FUNCTION_BLOCK HVAC_B28_Main_Seq
VAR_INPUT
END_VAR
VAR_OUTPUT
END_VAR
VAR
END_VAR

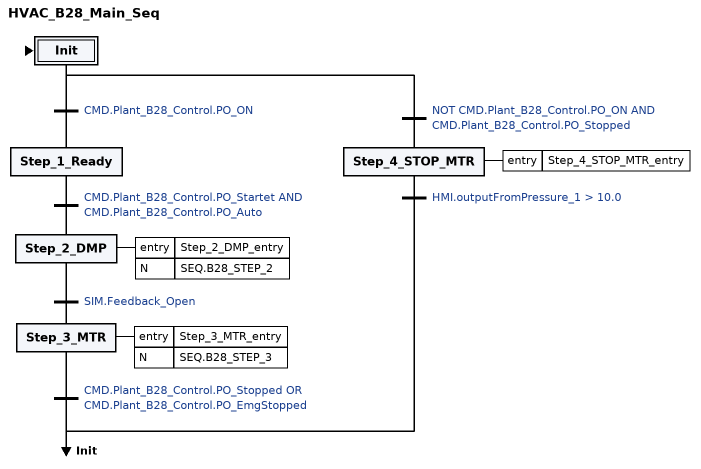
INITIAL_STEP Init:
END_STEP
TRANSITION FROM Init TO Step_1_Ready
    := CMD.Plant_B28_Control.PO_ON;
END_TRANSITION
STEP Step_1_Ready:
END_STEP
TRANSITION FROM Step_1_Ready TO Step_2_DMP
    := CMD.Plant_B28_Control.PO_Startet AND CMD.Plant_B28_Control.PO_Auto;
END_TRANSITION
STEP Step_2_DMP:
    Step_2_DMP_entry(P1);  // entry action
    SEQ.B28_STEP_2(N);
END_STEP
TRANSITION FROM Step_2_DMP TO Step_3_MTR
    := SIM.Feedback_Open;
END_TRANSITION
STEP Step_3_MTR:
    Step_3_MTR_entry(P1);  // entry action
    SEQ.B28_STEP_3(N);
END_STEP
TRANSITION FROM Step_3_MTR TO Init
    := CMD.Plant_B28_Control.PO_Stopped OR CMD.Plant_B28_Control.PO_EmgStopped;
END_TRANSITION
TRANSITION FROM Init TO Step_4_STOP_MTR
    := NOT CMD.Plant_B28_Control.PO_ON AND CMD.Plant_B28_Control.PO_Stopped;
END_TRANSITION
STEP Step_4_STOP_MTR:
    Step_4_STOP_MTR_entry(P1);  // entry action
END_STEP
TRANSITION FROM Step_4_STOP_MTR TO Init
    := HMI.outputFromPressure_1 > 10.0;
END_TRANSITION

ACTION Step_2_DMP_entry:
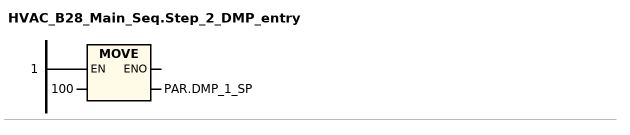
// NETWORK 1
PAR.DMP_1_SP := 100;
END_ACTION

ACTION Step_3_MTR_entry:
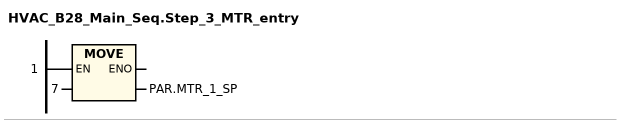
// NETWORK 1
PAR.MTR_1_SP := 7;
END_ACTION

ACTION Step_4_STOP_MTR_entry:
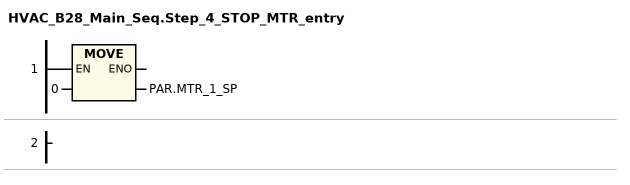
// NETWORK 1
PAR.MTR_1_SP := 0;

// NETWORK 2
END_ACTION

END_FUNCTION_BLOCK

(* stored: Version 1.1.0.1, ProductVersion 3.1.4024.13
   POU HVAC_B28_Main_Seq: Id {b5e85006-eed1-431b-ab11-5a9a7f0d6042}, SpecialFunc None
   Action Step_2_DMP_entry: Id {97ee2845-61bc-448e-8b0a-47fe686b2855}
   Action Step_3_MTR_entry: Id {cf48ad8c-42d2-4c93-9f4e-b2989cbbad3a}
   Action Step_4_STOP_MTR_entry: Id {787d6962-5456-4a74-9447-c9c39b81a23c} *)
